{attribute addProperty BoxType "EJ5002-0000-0017"}
{attribute addProperty Id "SSI_Inputs_ChannelAT %I*ARRAY[0..2] OF SSI_Inputs_Channel_32C7114D96120WcStateAT %I*WcState_98A4DF7520.250InfoDataAT %I*InfoData_BC63D37F80100"}
{attribute addProperty CRC "3984045230"}
{attribute addProperty SizeInBites "178"}
{attribute addProperty SizeInBytes "22.25"}
TYPE EJ5002_960CC6F1 :
STRUCT
	{attribute addProperty Name "SSI_Inputs_Channel"}
	SSI_Inputs_Channel : ARRAY[0..2] OF SSI_Inputs_Channel_32C7114D;
	{attribute addProperty Name "WcState"}
	WcState : WcState_98A4DF75;
	{attribute addProperty Name "InfoData"}
	InfoData : InfoData_BC63D37F;
END_STRUCT
END_TYPE

(* stored: Version 1.2.0.0, ProductVersion 3.1.4024.9
   DUT EJ5002_960CC6F1: Id {d997046e-760b-41d2-8936-583c7ce048d3} *)
